TYPE SoEReadProcessArgs :
STRUCT
	///SDO Index
	index: UINT;
	///Number of bytes to be read
	noOfBytes: UDINT;
END_STRUCT
END_TYPE

(* stored: Version 1.1.0.1, ProductVersion 3.1.4019.2
   DUT SoEReadProcessArgs: Id {5f6c0fef-11af-4996-a94f-3c169d4a0b75} *)
